   DropInserter.Drive.PLS.NotOperatorSide.HighLimit := 0.0;
   DropInserter.Drive.PLS.NotOperatorSide.Ok := FALSE;
   DropInserter.Drive.PLS.OnMould.LowLimit := 0.0;
   DropInserter.Drive.PLS.OnMould.HighLimit := 0.0;
   DropInserter.Drive.PLS.OnMould.Ok := FALSE;
   DropInserter.Drive.PLS.OffMould.LowLimit := 0.0;
   DropInserter.Drive.PLS.OffMould.HighLimit := 0.0;
   DropInserter.Drive.PLS.OffMould.Ok := FALSE;
   DropInserter.Drive.PLS.Pos0.LowLimit := 0.0;
   DropInserter.Drive.PLS.Pos0.HighLimit := 0.0;
   DropInserter.Drive.PLS.Pos0.Ok := FALSE;
   DropInserter.Drive.PLS.Pos1.LowLimit := 0.0;
   DropInserter.Drive.PLS.Pos1.HighLimit := 0.0;
   DropInserter.Drive.PLS.Pos1.Ok := FALSE;
   DropInserter.Drive.PLS.Pos2.LowLimit := 0.0;
   DropInserter.Drive.PLS.Pos2.HighLimit := 0.0;
   DropInserter.Drive.PLS.Pos2.Ok := FALSE;
   DropInserter.Drive.PLS.Pos3.LowLimit := 0.0;
   DropInserter.Drive.PLS.Pos3.HighLimit := 0.0;
   DropInserter.Drive.PLS.Pos3.Ok := FALSE;
   DropInserter.Drive.PLS.Pos4.LowLimit := 0.0;
   DropInserter.Drive.PLS.Pos4.HighLimit := 0.0;
   DropInserter.Drive.PLS.Pos4.Ok := FALSE;
   DropInserter.Drive.PLS.Pos5.LowLimit := 0.0;
   DropInserter.Drive.PLS.Pos5.HighLimit := 0.0;
   DropInserter.Drive.PLS.Pos5.Ok := FALSE;
   DropInserter.Drive.TON_EnableDrive.PT := T#500MS;
   DropInserter.Drive.TON_EnableDrive.IN := FALSE;
   DropInserter.Drive.TON_HwOvertravel_Dis.PT := T#0MS;
   DropInserter.Drive.TON_HwOvertravel_Dis.IN := FALSE;
   DropInserter.Drive.TON_HwOvertravel_En.PT := T#0MS;
   DropInserter.Drive.TON_HwOvertravel_En.IN := FALSE;
   DropInserter.Drive.TON_TimeoutMovement.PT := T#8S;
   DropInserter.Drive.TON_TimeoutMovement.IN := FALSE;
   DropInserter.TON_ResetMinLevel.PT := T#2S;
   DropInserter.TON_ResetMinLevel.IN := FALSE;
   DropInserter.RTO_Work.PT := T#1M;
   DropInserter.RTO_Work.IN := FALSE;
   DropInserter.TON_ScOK.PT := T#20S;
   DropInserter.TON_ScOK.IN := FALSE;
   DropInserter.TON_IncorrectPos.PT := T#2S;
   DropInserter.TON_IncorrectPos.IN := FALSE;
   DropInserter.TON_Sign_MinLevel.PT := T#1S;
   DropInserter.TON_Sign_MinLevel.IN := FALSE;
   DropInserter.TON_TimeoutWork.PT := T#20S;
   DropInserter.TON_TimeoutWork.IN := FALSE;
   DropInserter.TON_CloseCmd.PT := T#500MS;
   DropInserter.TON_CloseCmd.IN := FALSE;
   DropInserter.TON_MouldAbsence.PT := T#200MS;
   DropInserter.TON_MouldAbsence.IN := FALSE;
   PickInserter.ScOk := FALSE;
   PickInserter.CycleOn := FALSE;
   PickInserter.Work := FALSE;
   PickInserter.OkToStop := FALSE;
   PickInserter.AlmOk := TRUE;
   PickInserter.DrivesEnabled := FALSE;
   PickInserter.OutChainObstruction := FALSE;
   PickInserter.SingleCycle := FALSE;
   PickInserter.RepositioningReq := FALSE;
   PickInserter.Ons_TimeWork := FALSE;
   PickInserter.NumMinLevel := 0;
   PickInserter.Input.MouPreIns := FALSE;
   PickInserter.Input.EnaSel := FALSE;
   PickInserter.Input.MinLvl := FALSE;
   PickInserter.Input.HldCls := FALSE;
   PickInserter.Input.HldOpn := FALSE;
   PickInserter.Input.StrCls := FALSE;
   PickInserter.Input.StrOpn := FALSE;
   PickInserter.Output.EnaSelLgh := FALSE;
   PickInserter.Output.HldOpn := FALSE;
   PickInserter.Output.HldCls := FALSE;
   PickInserter.Output.StrOpn := FALSE;
   PickInserter.Output.StrCls := FALSE;
   PickInserter.Man.Ons_SingleCycle := FALSE;
   PickInserter.Man.CmdSupportOpen := FALSE;
   PickInserter.Man.CmdSupportClose := FALSE;
   PickInserter.Man.CmdStoreOpen := FALSE;
   PickInserter.Man.CmdStoreClose := FALSE;
   PickInserter.Man.CmdSingleCycle := FALSE;
   PickInserter.Man.EnaPbt := FALSE;
   PickInserter.Man.RstCmd := FALSE;
   PickInserter.Man.ScreenNumber := 302_080_301;
   PickInserter.Man.WithinScreenRange := 0;
   PickInserter."Step"._00_CycleActivated_DownCmd := FALSE;
   PickInserter."Step"._10_DownPos_OpenSupportCmd := FALSE;
   PickInserter."Step"._20_OpenSupportPos_CloseCmd := FALSE;
   PickInserter."Step"._30_ClosePos_CloseSupportCmd := FALSE;
   PickInserter."Step"._40_CloseSupportPos_UpCmd := FALSE;
   PickInserter."Step"._50_UpPos_OpenStoreCmd := FALSE;
   PickInserter."Step"._60_OpenStorePos_IntermediateCmd := FALSE;
   PickInserter."Step"._70_IntermediatePos_CloseStoreCmd := FALSE;
   PickInserter."Step"._80_CloseStorePos_CycleEnd := FALSE;
   PickInserter."Step".Ons_StrobeWorkDone := FALSE;
   PickInserter."Step".StrobeWorkDone := FALSE;
   PickInserter."Step".ScSeqOk := FALSE;
   PickInserter."Step".SeqActive := FALSE;
   PickInserter."Step".TON_WaitingHldOpn.PT := T#100MS;
   PickInserter."Step".TON_WaitingHldOpn.IN := FALSE;
   PickInserter."Step".TON_WaitingStrOpn.PT := T#100MS;
   PickInserter."Step".TON_WaitingStrOpn.IN := FALSE;
   PickInserter.Drive.AlmOk := FALSE;
   PickInserter.Drive.AlmEmerg := FALSE;
   PickInserter.Drive.AlmNode := FALSE;
   PickInserter.Drive.InitPosDrive := FALSE;
   PickInserter.Drive.InitPosDrivePLS := FALSE;
   PickInserter.Drive.GearingON := FALSE;
   PickInserter.Drive.CamHook := FALSE;
   PickInserter.Drive.CamStoppingPhase := FALSE;
   PickInserter.Drive.RepositioningRequest := FALSE;
   PickInserter.Drive.CamRequestResult := FALSE;
   PickInserter.Drive.CamRequestError := FALSE;
   PickInserter.Drive.CamRequestOk := FALSE;
   PickInserter.Drive.CalibDisAxisReq := FALSE;
   PickInserter.Drive.CalibReq := FALSE;
   PickInserter.Drive.CalibProcess := FALSE;
   PickInserter.Drive.HwOvertravelDisReq := FALSE;
   PickInserter.Drive.HwOvertravelEnReq := FALSE;
   PickInserter.Drive.AuxCamRequest := FALSE;
   PickInserter.Drive.TorquePeakEna := FALSE;
   PickInserter.Drive.Cmd_Repos := FALSE;
   PickInserter.Drive.Ons_CamRequest := FALSE;
   PickInserter.Drive.AuxCmdPosition := 0;
   PickInserter.Drive.Unwind := 0.0;
   PickInserter.Drive.MaxDev := 0.0;
   PickInserter.Drive.ReposSpeed := 100.0;
   PickInserter.Drive.CalcSlaveDifferenceABS := 0.0;
   PickInserter.Drive.CalcModPosition := 0.0;
   PickInserter.Drive.CalcSlaveDifference := 0.0;
   PickInserter.Drive.CalcMinDeltaPos := 0.0;
   PickInserter.Drive.CalcMaxDeltaPos := 0.0;
   PickInserter.Drive.CalcHalfPosUnwind := 0.0;
   PickInserter.Drive.Man.Cmd_PosJog := FALSE;
   PickInserter.Drive.Man.Cmd_NegJog := FALSE;
   PickInserter.Drive.Man.Cmd_Step := FALSE;
   PickInserter.Drive.Man.Cmd_Forward := FALSE;
   PickInserter.Drive.Man.Cmd_Backward := FALSE;
   PickInserter.Drive.Man.Cmd_Up := FALSE;
   PickInserter.Drive.Man.Cmd_Down := FALSE;
   PickInserter.Drive.Man.Cmd_Intermediate := FALSE;
   PickInserter.Drive.Man.Cmd_Open := FALSE;
   PickInserter.Drive.Man.Cmd_Close := FALSE;
   PickInserter.Drive.Man.Cmd_PreOpen := FALSE;
   PickInserter.Drive.Man.Cmd_Maintenance := FALSE;
   PickInserter.Drive.Man.Cmd_OperatorSide := FALSE;
   PickInserter.Drive.Man.Cmd_NotOperatorSide := FALSE;
   PickInserter.Drive.Man.Cmd_OnMould := FALSE;
   PickInserter.Drive.Man.Cmd_OffMould := FALSE;
   PickInserter.Drive.Man.Cmd_Pos0 := FALSE;
   PickInserter.Drive.Man.Cmd_Pos1 := FALSE;
   PickInserter.Drive.Man.Cmd_Pos2 := FALSE;
   PickInserter.Drive.Man.Cmd_Pos3 := FALSE;
   PickInserter.Drive.Man.Cmd_Pos4 := FALSE;
   PickInserter.Drive.Man.Cmd_Pos5 := FALSE;
   PickInserter.Drive.Man.Ons_Step := FALSE;
   PickInserter.Drive.Man.PhaseJogCmd := FALSE;
   PickInserter.Drive.Man.CmdStartStep := FALSE;
   PickInserter.Drive.Man.CmdEndStep := FALSE;
   PickInserter.Drive.Man.StepCond := FALSE;
   PickInserter.Drive.Man.TON_DelayHomeCmd.PT := T#3S;
   PickInserter.Drive.Man.TON_DelayHomeCmd.IN := FALSE;
   PickInserter.Drive.Auto.Cmd_Step := FALSE;
   PickInserter.Drive.Auto.Cmd_StartStep := FALSE;
   PickInserter.Drive.Auto.Cmd_EndStep := FALSE;
   PickInserter.Drive.Auto.Cmd_Forward := FALSE;
   PickInserter.Drive.Auto.Cmd_Backward := FALSE;
   PickInserter.Drive.Auto.Cmd_Up := FALSE;
   PickInserter.Drive.Auto.Cmd_Down := FALSE;
   PickInserter.Drive.Auto.Cmd_Intermediate := FALSE;
   PickInserter.Drive.Auto.Cmd_Open := FALSE;
   PickInserter.Drive.Auto.Cmd_Close := FALSE;
   PickInserter.Drive.Auto.Cmd_PreOpen := FALSE;
   PickInserter.Drive.Auto.Cmd_Maintenance := FALSE;
   PickInserter.Drive.Auto.Cmd_OperatorSide := FALSE;
   PickInserter.Drive.Auto.Cmd_NotOperatorSide := FALSE;
   PickInserter.Drive.Auto.Cmd_OnMould := FALSE;
   PickInserter.Drive.Auto.Cmd_OffMould := FALSE;
   PickInserter.Drive.Auto.Cmd_Pos0 := FALSE;
   PickInserter.Drive.Auto.Cmd_Pos1 := FALSE;
   PickInserter.Drive.Auto.Cmd_Pos2 := FALSE;
   PickInserter.Drive.Auto.Cmd_Pos3 := FALSE;
   PickInserter.Drive.Auto.Cmd_Pos4 := FALSE;
   PickInserter.Drive.Auto.Cmd_Pos5 := FALSE;
   PickInserter.Drive.Auto.Cmd_Gear := FALSE;
   PickInserter.Drive.ACT.CMD.Enable := FALSE;
   PickInserter.Drive.ACT.CMD.Pos_Mode := FALSE;
   PickInserter.Drive.ACT.CMD.MergeDisabled := FALSE;
   PickInserter.Drive.ACT.CMD.SCurve := FALSE;
   PickInserter.Drive.ACT.CMD.Cam_Mode := FALSE;
   PickInserter.Drive.ACT.CMD.Cam_Request := FALSE;
   PickInserter.Drive.ACT.CMD.Cam_PhaseStop := FALSE;
   PickInserter.Drive.ACT.CMD.Gear_Mode := FALSE;
   PickInserter.Drive.ACT.CMD.Repos_Req := FALSE;
   PickInserter.Drive.ACT.CMD.Jog_Pos := FALSE;
   PickInserter.Drive.ACT.CMD.Jog_Neg := FALSE;
   PickInserter.Drive.ACT.CMD.Stop := FALSE;
   PickInserter.Drive.ACT.CMD.Calibration_Req := FALSE;
   PickInserter.Drive.ACT.CMD.Reset := FALSE;
   PickInserter.Drive.ACT.CMD.RegInput1 := FALSE;
   PickInserter.Drive.ACT.CMD.Brake_Release := FALSE;
   PickInserter.Drive.ACT.CMD.HwPosOvertravel_Dis := FALSE;
   PickInserter.Drive.ACT.CMD.HwNegOvertravel_Dis := FALSE;
   PickInserter.Drive.ACT.CMD.HwOvertravel_MSG_En := FALSE;
   PickInserter.Drive.ACT.CMD.OneShootMove := FALSE;
   PickInserter.Drive.ACT.CMD.Move_Type := 0;
   PickInserter.Drive.ACT.CMD.Target_Pos := 0.0;
   PickInserter.Drive.ACT.CMD.Speed := 0.0;
   PickInserter.Drive.ACT.CMD.Acceleration := 0.0;
   PickInserter.Drive.ACT.CMD.Deceleration := 0.0;
   PickInserter.Drive.ACT.CMD.Torque_Limit := 0.0;
   PickInserter.Drive.ACT.CMD.Gear_Ratio := 0.0;
   PickInserter.Drive.ACT.CMD.Mccp_Length := 0;
   PickInserter.Drive.ACT.CMD.Mccp_StartSlope := 0.0;
   PickInserter.Drive.ACT.CMD.Mccp_EndSlope := 0.0;
   PickInserter.Drive.ACT.CMD.Mapc_Direction := 0;
   PickInserter.Drive.ACT.CMD.Mapc_SlaveScaling := 0.0;
   PickInserter.Drive.ACT.CMD.Mapc_MasterScaling := 0.0;
   PickInserter.Drive.ACT.CMD.Mapc_MasterLockPosition := 0.0;
   PickInserter.Drive.ACT.CMD.Mapc_CamLockPosition := 0.0;
   PickInserter.Drive.ACT.CMD.Cam[0..39].leadingValueStart := 0.0;
   PickInserter.Drive.ACT.CMD.Cam[0..39].leadingValueEnd := 0.0;
   PickInserter.Drive.ACT.CMD.Cam[0..39].followingValueStart := 0.0;
   PickInserter.Drive.ACT.CMD.Cam[0..39].followingValueEnd := 0.0;
   PickInserter.Drive.ACT.CMD.Cam[0..39].geoVeloStart := 0.0;
   PickInserter.Drive.ACT.CMD.Cam[0..39].geoVeloEnd := 0.0;
   PickInserter.Drive.ACT.CMD.Cam[0..39].geoAccelStart := 0.0;
   PickInserter.Drive.ACT.CMD.Cam[0..39].geoAccelEnd := 0.0;
   PickInserter.Drive.ACT.CMD.Cam[0..39].geoJerkStart := 0.0;
   PickInserter.Drive.ACT.CMD.Cam[0..39].geoJerkEnd := 0.0;
   PickInserter.Drive.ACT.CMD.Cam[0..39].inflectionPointParameter := 0.5;
   PickInserter.Drive.ACT.CMD.Cam[0..39].modVeloTrapezoidParameter := 1.0;
   PickInserter.Drive.ACT.CMD.Cam[0..39].modSineMaxAccelCaStar := 0.0;
   PickInserter.Drive.ACT.CMD.Cam[0..39].camProfileType := 0;
   PickInserter.Drive.ACT.FBK.Ready := FALSE;
   PickInserter.Drive.ACT.FBK.Calibrated := FALSE;
   PickInserter.Drive.ACT.FBK.Fault := FALSE;
   PickInserter.Drive.ACT.FBK.ModuleConnFault := FALSE;
   PickInserter.Drive.ACT.FBK.In_Position := FALSE;
   PickInserter.Drive.ACT.FBK.Standstill := FALSE;
   PickInserter.Drive.ACT.FBK.Enabled := FALSE;
   PickInserter.Drive.ACT.FBK.BusReadyStatus := FALSE;
   PickInserter.Drive.ACT.FBK.BrakeReleased := FALSE;
   PickInserter.Drive.ACT.FBK.HwPosOvertravelDisabled := FALSE;
   PickInserter.Drive.ACT.FBK.HwNegOvertravelDisabled := FALSE;
   PickInserter.Drive.ACT.FBK.SafeOffStatus := FALSE;
   PickInserter.Drive.ACT.FBK.MaxTorqueLimit := FALSE;
   PickInserter.Drive.ACT.FBK.PosMerge_IP := FALSE;
   PickInserter.Drive.ACT.FBK.PosMerge_PC := FALSE;
   PickInserter.Drive.ACT.FBK.Gearing_IP := FALSE;
   PickInserter.Drive.ACT.FBK.Position := 0.0;
   PickInserter.Drive.ACT.FBK.Speed := 0.0;
   PickInserter.Drive.ACT.FBK.Torque := 0.0;
   PickInserter.Drive.ACT.FBK.RegInput1Pos := 0.0;
   PickInserter.Drive.ACT.FBK.SeqCamErrorCode := 0;
   PickInserter.Drive.ACT.FBK.SeqCamTargetPosMAM := 0.0;
   PickInserter.Drive.ACT.FBK.SeqCamStatus.EndSequence := FALSE;
   PickInserter.Drive.ACT.FBK.SeqCamStatus.EndSuccess := FALSE;
   PickInserter.Drive.ACT.FBK.SeqCamStatus.EndError := FALSE;
   PickInserter.Drive.ACT.FBK.SeqCamStatus.CamHook := FALSE;
   PickInserter.Drive.ACT.FBK.SeqCamStatus.BothMapc_IP := FALSE;
   PickInserter.Drive.ACT.FBK.SeqCamStatus.SlaveFwd := FALSE;
   PickInserter.Drive.ACT.FBK.SeqCamStatus.SlaveBwd := FALSE;
   PickInserter.Drive.ACT.FBK.SeqCamStatus.SlaveUnwind := FALSE;
   PickInserter.Drive.ACT.FBK.SeqCamStatus.WaitValidByOpe := FALSE;
   PickInserter.Drive.ACT.FBK.SeqCamStatus.MapcA_IP := FALSE;
   PickInserter.Drive.ACT.FBK.SeqCamStatus.MapcB_IP := FALSE;
   PickInserter.Drive.ACT.FBK.SeqCamStatus.MapcC_IP := FALSE;
   PickInserter.Drive.ACT.FBK.SeqCamStatus.CamOnce_PC := FALSE;
   PickInserter.Drive.ACT.FBK.SeqCamStatus.MaxDevError := FALSE;
   PickInserter.Drive.ACT.FBK.SeqCamStatus.PositionCamLockStatus := FALSE;
   PickInserter.Drive.ACT.FBK.SeqCamStatus.WaitRestart := FALSE;
   PickInserter.Drive.ACT.FBK.SeqCamStatus.Bit17 := FALSE;
   PickInserter.Drive.ACT.FBK.SeqCamStatus.Bit18 := FALSE;
   PickInserter.Drive.ACT.FBK.SeqCamStatus.Bit19 := FALSE;
   PickInserter.Drive.ACT.FBK.SeqCamStatus.Bit20 := FALSE;
   PickInserter.Drive.ACT.FBK.SeqCamStatus.Bit21 := FALSE;
   PickInserter.Drive.ACT.FBK.SeqCamStatus.Bit22 := FALSE;
   PickInserter.Drive.ACT.FBK.SeqCamStatus.Bit23 := FALSE;
   PickInserter.Drive.ACT.FBK.SeqCamStatus.Bit24 := FALSE;
   PickInserter.Drive.ACT.FBK.SeqCamStatus.Bit25 := FALSE;
   PickInserter.Drive.ACT.FBK.SeqCamStatus.Bit26 := FALSE;
   PickInserter.Drive.ACT.FBK.SeqCamStatus.Bit27 := FALSE;
   PickInserter.Drive.ACT.FBK.SeqCamStatus.Bit28 := FALSE;
   PickInserter.Drive.ACT.FBK.SeqCamStatus.Bit29 := FALSE;
   PickInserter.Drive.ACT.FBK.SeqCamStatus.Bit30 := FALSE;
   PickInserter.Drive.ACT.FBK.SeqCamStatus.Bit31 := FALSE;
   PickInserter.Drive.ACT.FBK.SeqCamStatus.Bit32 := FALSE;
   PickInserter.Drive.PLS.FinePosOk.LowLimit := 0.0;
   PickInserter.Drive.PLS.FinePosOk.HighLimit := 0.0;
   PickInserter.Drive.PLS.FinePosOk.Ok := FALSE;
   PickInserter.Drive.PLS.KeepPosOk.LowLimit := 0.0;
   PickInserter.Drive.PLS.KeepPosOk.HighLimit := 0.0;
   PickInserter.Drive.PLS.KeepPosOk.Ok := FALSE;
   PickInserter.Drive.PLS.Up.LowLimit := 0.0;
   PickInserter.Drive.PLS.Up.HighLimit := 0.0;
   PickInserter.Drive.PLS.Up.Ok := FALSE;
   PickInserter.Drive.PLS.Intermediate.LowLimit := 0.0;
   PickInserter.Drive.PLS.Intermediate.HighLimit := 0.0;
   PickInserter.Drive.PLS.Intermediate.Ok := FALSE;
   PickInserter.Drive.PLS.Down.LowLimit := 0.0;
   PickInserter.Drive.PLS.Down.HighLimit := 0.0;
   PickInserter.Drive.PLS.Down.Ok := FALSE;
   PickInserter.Drive.PLS.Forward.LowLimit := 0.0;
   PickInserter.Drive.PLS.Forward.HighLimit := 0.0;
   PickInserter.Drive.PLS.Forward.Ok := FALSE;
   PickInserter.Drive.PLS.Backward.LowLimit := 0.0;
   PickInserter.Drive.PLS.Backward.HighLimit := 0.0;
   PickInserter.Drive.PLS.Backward.Ok := FALSE;
   PickInserter.Drive.PLS.Open.LowLimit := 0.0;
   PickInserter.Drive.PLS.Open.HighLimit := 0.0;
   PickInserter.Drive.PLS.Open.Ok := FALSE;
   PickInserter.Drive.PLS.Close.LowLimit := 0.0;
   PickInserter.Drive.PLS.Close.HighLimit := 0.0;
   PickInserter.Drive.PLS.Close.Ok := FALSE;
   PickInserter.Drive.PLS.PreOpen.LowLimit := 0.0;
   PickInserter.Drive.PLS.PreOpen.HighLimit := 0.0;
   PickInserter.Drive.PLS.PreOpen.Ok := FALSE;
   PickInserter.Drive.PLS.Maintenance.LowLimit := 0.0;
   PickInserter.Drive.PLS.Maintenance.HighLimit := 0.0;
   PickInserter.Drive.PLS.Maintenance.Ok := FALSE;
   PickInserter.Drive.PLS.OperatorSide.LowLimit := 0.0;
   PickInserter.Drive.PLS.OperatorSide.HighLimit := 0.0;
   PickInserter.Drive.PLS.OperatorSide.Ok := FALSE;
   PickInserter.Drive.PLS.NotOperatorSide.LowLimit := 0.0;
   PickInserter.Drive.PLS.NotOperatorSide.HighLimit := 0.0;
   PickInserter.Drive.PLS.NotOperatorSide.Ok := FALSE;
   PickInserter.Drive.PLS.OnMould.LowLimit := 0.0;
   PickInserter.Drive.PLS.OnMould.HighLimit := 0.0;
   PickInserter.Drive.PLS.OnMould.Ok := FALSE;
   PickInserter.Drive.PLS.OffMould.LowLimit := 0.0;
   PickInserter.Drive.PLS.OffMould.HighLimit := 0.0;
   PickInserter.Drive.PLS.OffMould.Ok := FALSE;
   PickInserter.Drive.PLS.Pos0.LowLimit := 0.0;
   PickInserter.Drive.PLS.Pos0.HighLimit := 0.0;
   PickInserter.Drive.PLS.Pos0.Ok := FALSE;
   PickInserter.Drive.PLS.Pos1.LowLimit := 0.0;
   PickInserter.Drive.PLS.Pos1.HighLimit := 0.0;
   PickInserter.Drive.PLS.Pos1.Ok := FALSE;
   PickInserter.Drive.PLS.Pos2.LowLimit := 0.0;
   PickInserter.Drive.PLS.Pos2.HighLimit := 0.0;
   PickInserter.Drive.PLS.Pos2.Ok := FALSE;
   PickInserter.Drive.PLS.Pos3.LowLimit := 0.0;
   PickInserter.Drive.PLS.Pos3.HighLimit := 0.0;
   PickInserter.Drive.PLS.Pos3.Ok := FALSE;
   PickInserter.Drive.PLS.Pos4.LowLimit := 0.0;
   PickInserter.Drive.PLS.Pos4.HighLimit := 0.0;
   PickInserter.Drive.PLS.Pos4.Ok := FALSE;
   PickInserter.Drive.PLS.Pos5.LowLimit := 0.0;
   PickInserter.Drive.PLS.Pos5.HighLimit := 0.0;
   PickInserter.Drive.PLS.Pos5.Ok := FALSE;
   PickInserter.Drive.TON_EnableDrive.PT := T#500MS;
   PickInserter.Drive.TON_EnableDrive.IN := FALSE;
   PickInserter.Drive.TON_HwOvertravel_Dis.PT := T#0MS;
   PickInserter.Drive.TON_HwOvertravel_Dis.IN := FALSE;
   PickInserter.Drive.TON_HwOvertravel_En.PT := T#0MS;
   PickInserter.Drive.TON_HwOvertravel_En.IN := FALSE;
   PickInserter.Drive.TON_TimeoutMovement.PT := T#8S;
   PickInserter.Drive.TON_TimeoutMovement.IN := FALSE;
   PickInserter.TON_ResetMinLevel.PT := T#2S;
   PickInserter.TON_ResetMinLevel.IN := FALSE;
   PickInserter.RTO_Work.PT := T#1M;
   PickInserter.RTO_Work.IN := FALSE;
   PickInserter.TON_ScOK.PT := T#20S;
   PickInserter.TON_ScOK.IN := FALSE;
   PickInserter.TON_SupportIncorrectPos.PT := T#2S;
   PickInserter.TON_SupportIncorrectPos.IN := FALSE;
   PickInserter.TON_StoreIncorrectPos.PT := T#2S;
   PickInserter.TON_StoreIncorrectPos.IN := FALSE;
   PickInserter.TON_Sign_MinLevel.PT := T#1S;
   PickInserter.TON_Sign_MinLevel.IN := FALSE;
   PickInserter.TON_TimeoutWork.PT := T#20S;
   PickInserter.TON_TimeoutWork.IN := FALSE;
   PickInserter.TON_MouldAbsence.PT := T#200MS;
   PickInserter.TON_MouldAbsence.IN := FALSE;
   RotaryInserter.ScOk := FALSE;
   RotaryInserter.CycleOn := FALSE;
   RotaryInserter.Work := FALSE;
   RotaryInserter.OkToStop := TRUE;
   RotaryInserter.AlmOk := TRUE;
   RotaryInserter.DrivesEnabled := FALSE;
   RotaryInserter.OutChainObstruction := TRUE;
   RotaryInserter.RepositioningReq := FALSE;
   RotaryInserter.Ons_TimeWork := TRUE;
   RotaryInserter.NumMinLevel := 0;
   RotaryInserter.Input.MouPreIns := TRUE;
   RotaryInserter.Input.EnaSel := FALSE;
   RotaryInserter.Input.MinLvl := TRUE;
   RotaryInserter.Output.EnaSelLgh := FALSE;
   RotaryInserter.Man.EnaPbt := FALSE;
   RotaryInserter.Man.RstCmd := TRUE;
   RotaryInserter.Man.ScreenNumber := 302_090_301;
   RotaryInserter.Man.WithinScreenRange := 0;
   RotaryInserter."Step"._00_CycleActived_StartRotationCmd := FALSE;
   RotaryInserter."Step"._10_RotationOutPos_StopRotationCmd := FALSE;
   RotaryInserter."Step"._20_FinePos_IncreaseMinLevMouCmd := FALSE;
   RotaryInserter."Step"._30_MinLevInc_CycleEnd := FALSE;
   RotaryInserter."Step".Ons_StrobeWorkDone := FALSE;
   RotaryInserter."Step".StrobeWorkDone := FALSE;
   RotaryInserter."Step".ScSeqOk := FALSE;
   RotaryInserter."Step".SeqActive := FALSE;
   RotaryInserter.Drive.AlmOk := FALSE;
   RotaryInserter.Drive.AlmEmerg := FALSE;
   RotaryInserter.Drive.AlmNode := FALSE;
   RotaryInserter.Drive.InitPosDrive := FALSE;
   RotaryInserter.Drive.InitPosDrivePLS := FALSE;
   RotaryInserter.Drive.GearingON := FALSE;
   RotaryInserter.Drive.CamHook := FALSE;
   RotaryInserter.Drive.CamStoppingPhase := FALSE;
   RotaryInserter.Drive.RepositioningRequest := FALSE;
   RotaryInserter.Drive.CamRequestResult := FALSE;
   RotaryInserter.Drive.CamRequestError := FALSE;
   RotaryInserter.Drive.CamRequestOk := FALSE;
   RotaryInserter.Drive.CalibDisAxisReq := FALSE;
   RotaryInserter.Drive.CalibReq := FALSE;
   RotaryInserter.Drive.CalibProcess := FALSE;
   RotaryInserter.Drive.HwOvertravelDisReq := FALSE;
   RotaryInserter.Drive.HwOvertravelEnReq := FALSE;
   RotaryInserter.Drive.AuxCamRequest := FALSE;
   RotaryInserter.Drive.TorquePeakEna := TRUE;
   RotaryInserter.Drive.Cmd_Repos := FALSE;
   RotaryInserter.Drive.Ons_CamRequest := FALSE;
   RotaryInserter.Drive.AuxCmdPosition := 0;
   RotaryInserter.Drive.Unwind := 360.0;
   RotaryInserter.Drive.MaxDev := 0.0;
   RotaryInserter.Drive.ReposSpeed := 100.0;
   RotaryInserter.Drive.CalcSlaveDifferenceABS := 0.0;
   RotaryInserter.Drive.CalcModPosition := 0.0;
   RotaryInserter.Drive.CalcSlaveDifference := 0.0;
   RotaryInserter.Drive.CalcMinDeltaPos := 0.0;
   RotaryInserter.Drive.CalcMaxDeltaPos := 0.0;
   RotaryInserter.Drive.CalcHalfPosUnwind := 0.0;
   RotaryInserter.Drive.Man.Cmd_PosJog := FALSE;
   RotaryInserter.Drive.Man.Cmd_NegJog := FALSE;
   RotaryInserter.Drive.Man.Cmd_Step := FALSE;
   RotaryInserter.Drive.Man.Cmd_Forward := FALSE;
   RotaryInserter.Drive.Man.Cmd_Backward := FALSE;
   RotaryInserter.Drive.Man.Cmd_Up := FALSE;
   RotaryInserter.Drive.Man.Cmd_Down := FALSE;
   RotaryInserter.Drive.Man.Cmd_Intermediate := FALSE;
   RotaryInserter.Drive.Man.Cmd_Open := FALSE;
   RotaryInserter.Drive.Man.Cmd_Close := FALSE;
   RotaryInserter.Drive.Man.Cmd_PreOpen := FALSE;
   RotaryInserter.Drive.Man.Cmd_Maintenance := FALSE;
   RotaryInserter.Drive.Man.Cmd_OperatorSide := FALSE;
   RotaryInserter.Drive.Man.Cmd_NotOperatorSide := FALSE;
   RotaryInserter.Drive.Man.Cmd_OnMould := FALSE;
   RotaryInserter.Drive.Man.Cmd_OffMould := FALSE;
   RotaryInserter.Drive.Man.Cmd_Pos0 := FALSE;
   RotaryInserter.Drive.Man.Cmd_Pos1 := FALSE;
   RotaryInserter.Drive.Man.Cmd_Pos2 := FALSE;
   RotaryInserter.Drive.Man.Cmd_Pos3 := FALSE;
   RotaryInserter.Drive.Man.Cmd_Pos4 := FALSE;
   RotaryInserter.Drive.Man.Cmd_Pos5 := FALSE;
   RotaryInserter.Drive.Man.Ons_Step := FALSE;
   RotaryInserter.Drive.Man.PhaseJogCmd := FALSE;
   RotaryInserter.Drive.Man.CmdStartStep := FALSE;
   RotaryInserter.Drive.Man.CmdEndStep := FALSE;
   RotaryInserter.Drive.Man.StepCond := FALSE;
   RotaryInserter.Drive.Man.TON_DelayHomeCmd.PT := T#3S;
   RotaryInserter.Drive.Man.TON_DelayHomeCmd.IN := FALSE;
   RotaryInserter.Drive.Auto.Cmd_Step := FALSE;
   RotaryInserter.Drive.Auto.Cmd_StartStep := FALSE;
   RotaryInserter.Drive.Auto.Cmd_EndStep := FALSE;
   RotaryInserter.Drive.Auto.Cmd_Forward := FALSE;
   RotaryInserter.Drive.Auto.Cmd_Backward := FALSE;
   RotaryInserter.Drive.Auto.Cmd_Up := FALSE;
   RotaryInserter.Drive.Auto.Cmd_Down := FALSE;
   RotaryInserter.Drive.Auto.Cmd_Intermediate := FALSE;
   RotaryInserter.Drive.Auto.Cmd_Open := FALSE;
   RotaryInserter.Drive.Auto.Cmd_Close := FALSE;
   RotaryInserter.Drive.Auto.Cmd_PreOpen := FALSE;
   RotaryInserter.Drive.Auto.Cmd_Maintenance := FALSE;
   RotaryInserter.Drive.Auto.Cmd_OperatorSide := FALSE;
   RotaryInserter.Drive.Auto.Cmd_NotOperatorSide := FALSE;
   RotaryInserter.Drive.Auto.Cmd_OnMould := FALSE;
   RotaryInserter.Drive.Auto.Cmd_OffMould := FALSE;
   RotaryInserter.Drive.Auto.Cmd_Pos0 := FALSE;
   RotaryInserter.Drive.Auto.Cmd_Pos1 := FALSE;
   RotaryInserter.Drive.Auto.Cmd_Pos2 := FALSE;
   RotaryInserter.Drive.Auto.Cmd_Pos3 := FALSE;
   RotaryInserter.Drive.Auto.Cmd_Pos4 := FALSE;
   RotaryInserter.Drive.Auto.Cmd_Pos5 := FALSE;
   RotaryInserter.Drive.Auto.Cmd_Gear := FALSE;
   RotaryInserter.Drive.ACT.CMD.Enable := FALSE;
   RotaryInserter.Drive.ACT.CMD.Pos_Mode := FALSE;
   RotaryInserter.Drive.ACT.CMD.MergeDisabled := FALSE;
   RotaryInserter.Drive.ACT.CMD.SCurve := FALSE;
   RotaryInserter.Drive.ACT.CMD.Cam_Mode := FALSE;
   RotaryInserter.Drive.ACT.CMD.Cam_Request := FALSE;
   RotaryInserter.Drive.ACT.CMD.Cam_PhaseStop := FALSE;
   RotaryInserter.Drive.ACT.CMD.Gear_Mode := FALSE;
   RotaryInserter.Drive.ACT.CMD.Repos_Req := FALSE;
   RotaryInserter.Drive.ACT.CMD.Jog_Pos := FALSE;
   RotaryInserter.Drive.ACT.CMD.Jog_Neg := FALSE;
   RotaryInserter.Drive.ACT.CMD.Stop := TRUE;
   RotaryInserter.Drive.ACT.CMD.Calibration_Req := FALSE;
   RotaryInserter.Drive.ACT.CMD.Reset := FALSE;
   RotaryInserter.Drive.ACT.CMD.RegInput1 := FALSE;
   RotaryInserter.Drive.ACT.CMD.Brake_Release := FALSE;
   RotaryInserter.Drive.ACT.CMD.HwPosOvertravel_Dis := FALSE;
   RotaryInserter.Drive.ACT.CMD.HwNegOvertravel_Dis := FALSE;
   RotaryInserter.Drive.ACT.CMD.HwOvertravel_MSG_En := FALSE;
   RotaryInserter.Drive.ACT.CMD.OneShootMove := FALSE;
   RotaryInserter.Drive.ACT.CMD.Move_Type := 3;
   RotaryInserter.Drive.ACT.CMD.Target_Pos := 0.0;
   RotaryInserter.Drive.ACT.CMD.Speed := 250.0;
   RotaryInserter.Drive.ACT.CMD.Acceleration := 4000.0;
   RotaryInserter.Drive.ACT.CMD.Deceleration := 4500.0;
   RotaryInserter.Drive.ACT.CMD.Torque_Limit := 50.0;
   RotaryInserter.Drive.ACT.CMD.Gear_Ratio := 0.0;
   RotaryInserter.Drive.ACT.CMD.Mccp_Length := 0;
   RotaryInserter.Drive.ACT.CMD.Mccp_StartSlope := 0.0;
   RotaryInserter.Drive.ACT.CMD.Mccp_EndSlope := 0.0;
   RotaryInserter.Drive.ACT.CMD.Mapc_Direction := 0;
   RotaryInserter.Drive.ACT.CMD.Mapc_SlaveScaling := 0.0;
   RotaryInserter.Drive.ACT.CMD.Mapc_MasterScaling := 0.0;
   RotaryInserter.Drive.ACT.CMD.Mapc_MasterLockPosition := 0.0;
   RotaryInserter.Drive.ACT.CMD.Mapc_CamLockPosition := 0.0;
   RotaryInserter.Drive.ACT.CMD.Cam[0..39].leadingValueStart := 0.0;
   RotaryInserter.Drive.ACT.CMD.Cam[0..39].leadingValueEnd := 0.0;
   RotaryInserter.Drive.ACT.CMD.Cam[0..39].followingValueStart := 0.0;
   RotaryInserter.Drive.ACT.CMD.Cam[0..39].followingValueEnd := 0.0;
   RotaryInserter.Drive.ACT.CMD.Cam[0..39].geoVeloStart := 0.0;
   RotaryInserter.Drive.ACT.CMD.Cam[0..39].geoVeloEnd := 0.0;
   RotaryInserter.Drive.ACT.CMD.Cam[0..39].geoAccelStart := 0.0;
   RotaryInserter.Drive.ACT.CMD.Cam[0..39].geoAccelEnd := 0.0;
   RotaryInserter.Drive.ACT.CMD.Cam[0..39].geoJerkStart := 0.0;
   RotaryInserter.Drive.ACT.CMD.Cam[0..39].geoJerkEnd := 0.0;
   RotaryInserter.Drive.ACT.CMD.Cam[0..39].inflectionPointParameter := 0.5;
   RotaryInserter.Drive.ACT.CMD.Cam[0..39].modVeloTrapezoidParameter := 1.0;
   RotaryInserter.Drive.ACT.CMD.Cam[0..39].modSineMaxAccelCaStar := 0.0;
   RotaryInserter.Drive.ACT.CMD.Cam[0..39].camProfileType := 0;
   RotaryInserter.Drive.ACT.FBK.Ready := TRUE;
   RotaryInserter.Drive.ACT.FBK.Calibrated := TRUE;
   RotaryInserter.Drive.ACT.FBK.Fault := FALSE;
   RotaryInserter.Drive.ACT.FBK.ModuleConnFault := FALSE;
   RotaryInserter.Drive.ACT.FBK.In_Position := FALSE;
   RotaryInserter.Drive.ACT.FBK.Standstill := TRUE;
   RotaryInserter.Drive.ACT.FBK.Enabled := FALSE;
   RotaryInserter.Drive.ACT.FBK.BusReadyStatus := FALSE;
   RotaryInserter.Drive.ACT.FBK.BrakeReleased := FALSE;
   RotaryInserter.Drive.ACT.FBK.HwPosOvertravelDisabled := FALSE;
   RotaryInserter.Drive.ACT.FBK.HwNegOvertravelDisabled := FALSE;
   RotaryInserter.Drive.ACT.FBK.SafeOffStatus := FALSE;
   RotaryInserter.Drive.ACT.FBK.MaxTorqueLimit := FALSE;
   RotaryInserter.Drive.ACT.FBK.PosMerge_IP := FALSE;
   RotaryInserter.Drive.ACT.FBK.PosMerge_PC := FALSE;
   RotaryInserter.Drive.ACT.FBK.Gearing_IP := FALSE;
   RotaryInserter.Drive.ACT.FBK.Position := 0.81;
   RotaryInserter.Drive.ACT.FBK.Speed := -0.02503395;
   RotaryInserter.Drive.ACT.FBK.Torque := 0.0;
   RotaryInserter.Drive.ACT.FBK.RegInput1Pos := 0.0;
   RotaryInserter.Drive.ACT.FBK.SeqCamErrorCode := 0;
   RotaryInserter.Drive.ACT.FBK.SeqCamTargetPosMAM := 0.0;
   RotaryInserter.Drive.ACT.FBK.SeqCamStatus.EndSequence := FALSE;
   RotaryInserter.Drive.ACT.FBK.SeqCamStatus.EndSuccess := FALSE;
   RotaryInserter.Drive.ACT.FBK.SeqCamStatus.EndError := FALSE;
   RotaryInserter.Drive.ACT.FBK.SeqCamStatus.CamHook := FALSE;
   RotaryInserter.Drive.ACT.FBK.SeqCamStatus.BothMapc_IP := FALSE;
   RotaryInserter.Drive.ACT.FBK.SeqCamStatus.SlaveFwd := FALSE;
   RotaryInserter.Drive.ACT.FBK.SeqCamStatus.SlaveBwd := FALSE;
   RotaryInserter.Drive.ACT.FBK.SeqCamStatus.SlaveUnwind := FALSE;
   RotaryInserter.Drive.ACT.FBK.SeqCamStatus.WaitValidByOpe := FALSE;
   RotaryInserter.Drive.ACT.FBK.SeqCamStatus.MapcA_IP := FALSE;
   RotaryInserter.Drive.ACT.FBK.SeqCamStatus.MapcB_IP := FALSE;
   RotaryInserter.Drive.ACT.FBK.SeqCamStatus.MapcC_IP := FALSE;
   RotaryInserter.Drive.ACT.FBK.SeqCamStatus.CamOnce_PC := FALSE;
   RotaryInserter.Drive.ACT.FBK.SeqCamStatus.MaxDevError := FALSE;
   RotaryInserter.Drive.ACT.FBK.SeqCamStatus.PositionCamLockStatus := FALSE;
   RotaryInserter.Drive.ACT.FBK.SeqCamStatus.WaitRestart := FALSE;
   RotaryInserter.Drive.ACT.FBK.SeqCamStatus.Bit17 := FALSE;
   RotaryInserter.Drive.ACT.FBK.SeqCamStatus.Bit18 := FALSE;
   RotaryInserter.Drive.ACT.FBK.SeqCamStatus.Bit19 := FALSE;
   RotaryInserter.Drive.ACT.FBK.SeqCamStatus.Bit20 := FALSE;
   RotaryInserter.Drive.ACT.FBK.SeqCamStatus.Bit21 := FALSE;
   RotaryInserter.Drive.ACT.FBK.SeqCamStatus.Bit22 := FALSE;
   RotaryInserter.Drive.ACT.FBK.SeqCamStatus.Bit23 := FALSE;
   RotaryInserter.Drive.ACT.FBK.SeqCamStatus.Bit24 := FALSE;
   RotaryInserter.Drive.ACT.FBK.SeqCamStatus.Bit25 := FALSE;
   RotaryInserter.Drive.ACT.FBK.SeqCamStatus.Bit26 := FALSE;
   RotaryInserter.Drive.ACT.FBK.SeqCamStatus.Bit27 := FALSE;
   RotaryInserter.Drive.ACT.FBK.SeqCamStatus.Bit28 := FALSE;
   RotaryInserter.Drive.ACT.FBK.SeqCamStatus.Bit29 := FALSE;
   RotaryInserter.Drive.ACT.FBK.SeqCamStatus.Bit30 := FALSE;
   RotaryInserter.Drive.ACT.FBK.SeqCamStatus.Bit31 := FALSE;
   RotaryInserter.Drive.ACT.FBK.SeqCamStatus.Bit32 := FALSE;
   RotaryInserter.Drive.PLS.FinePosOk.LowLimit := 357.0;
   RotaryInserter.Drive.PLS.FinePosOk.HighLimit := 3.0;
   RotaryInserter.Drive.PLS.FinePosOk.Ok := TRUE;
   RotaryInserter.Drive.PLS.KeepPosOk.LowLimit := 0.0;
   RotaryInserter.Drive.PLS.KeepPosOk.HighLimit := 0.0;
   RotaryInserter.Drive.PLS.KeepPosOk.Ok := FALSE;
   RotaryInserter.Drive.PLS.Up.LowLimit := 0.0;
   RotaryInserter.Drive.PLS.Up.HighLimit := 0.0;
   RotaryInserter.Drive.PLS.Up.Ok := FALSE;
   RotaryInserter.Drive.PLS.Intermediate.LowLimit := 0.0;
   RotaryInserter.Drive.PLS.Intermediate.HighLimit := 0.0;
   RotaryInserter.Drive.PLS.Intermediate.Ok := FALSE;
   RotaryInserter.Drive.PLS.Down.LowLimit := 0.0;
   RotaryInserter.Drive.PLS.Down.HighLimit := 0.0;
   RotaryInserter.Drive.PLS.Down.Ok := FALSE;
   RotaryInserter.Drive.PLS.Forward.LowLimit := 0.0;
   RotaryInserter.Drive.PLS.Forward.HighLimit := 0.0;
   RotaryInserter.Drive.PLS.Forward.Ok := FALSE;
   RotaryInserter.Drive.PLS.Backward.LowLimit := 0.0;
   RotaryInserter.Drive.PLS.Backward.HighLimit := 0.0;
   RotaryInserter.Drive.PLS.Backward.Ok := FALSE;
   RotaryInserter.Drive.PLS.Open.LowLimit := 0.0;
   RotaryInserter.Drive.PLS.Open.HighLimit := 0.0;
   RotaryInserter.Drive.PLS.Open.Ok := FALSE;
   RotaryInserter.Drive.PLS.Close.LowLimit := 0.0;
   RotaryInserter.Drive.PLS.Close.HighLimit := 0.0;
   RotaryInserter.Drive.PLS.Close.Ok := FALSE;
   RotaryInserter.Drive.PLS.PreOpen.LowLimit := 0.0;
   RotaryInserter.Drive.PLS.PreOpen.HighLimit := 0.0;
   RotaryInserter.Drive.PLS.PreOpen.Ok := FALSE;
   RotaryInserter.Drive.PLS.Maintenance.LowLimit := 0.0;
   RotaryInserter.Drive.PLS.Maintenance.HighLimit := 0.0;
   RotaryInserter.Drive.PLS.Maintenance.Ok := FALSE;
   RotaryInserter.Drive.PLS.OperatorSide.LowLimit := 0.0;
   RotaryInserter.Drive.PLS.OperatorSide.HighLimit := 0.0;
   RotaryInserter.Drive.PLS.OperatorSide.Ok := FALSE;
   RotaryInserter.Drive.PLS.NotOperatorSide.LowLimit := 0.0;
   RotaryInserter.Drive.PLS.NotOperatorSide.HighLimit := 0.0;
   RotaryInserter.Drive.PLS.NotOperatorSide.Ok := FALSE;
   RotaryInserter.Drive.PLS.OnMould.LowLimit := 0.0;
   RotaryInserter.Drive.PLS.OnMould.HighLimit := 0.0;
   RotaryInserter.Drive.PLS.OnMould.Ok := FALSE;
   RotaryInserter.Drive.PLS.OffMould.LowLimit := 0.0;
   RotaryInserter.Drive.PLS.OffMould.HighLimit := 0.0;
   RotaryInserter.Drive.PLS.OffMould.Ok := FALSE;
   RotaryInserter.Drive.PLS.Pos0.LowLimit := 0.0;
   RotaryInserter.Drive.PLS.Pos0.HighLimit := 0.0;
   RotaryInserter.Drive.PLS.Pos0.Ok := FALSE;
   RotaryInserter.Drive.PLS.Pos1.LowLimit := 0.0;
   RotaryInserter.Drive.PLS.Pos1.HighLimit := 0.0;
   RotaryInserter.Drive.PLS.Pos1.Ok := FALSE;
   RotaryInserter.Drive.PLS.Pos2.LowLimit := 0.0;
   RotaryInserter.Drive.PLS.Pos2.HighLimit := 0.0;
   RotaryInserter.Drive.PLS.Pos2.Ok := FALSE;
   RotaryInserter.Drive.PLS.Pos3.LowLimit := 0.0;
   RotaryInserter.Drive.PLS.Pos3.HighLimit := 0.0;
   RotaryInserter.Drive.PLS.Pos3.Ok := FALSE;
   RotaryInserter.Drive.PLS.Pos4.LowLimit := 0.0;
   RotaryInserter.Drive.PLS.Pos4.HighLimit := 0.0;
   RotaryInserter.Drive.PLS.Pos4.Ok := FALSE;
   RotaryInserter.Drive.PLS.Pos5.LowLimit := 0.0;
   RotaryInserter.Drive.PLS.Pos5.HighLimit := 0.0;
   RotaryInserter.Drive.PLS.Pos5.Ok := FALSE;
   RotaryInserter.Drive.TON_EnableDrive.PT := T#500MS;
   RotaryInserter.Drive.TON_EnableDrive.IN := FALSE;
   RotaryInserter.Drive.TON_HwOvertravel_Dis.PT := T#0MS;
   RotaryInserter.Drive.TON_HwOvertravel_Dis.IN := FALSE;
   RotaryInserter.Drive.TON_HwOvertravel_En.PT := T#0MS;
   RotaryInserter.Drive.TON_HwOvertravel_En.IN := FALSE;
   RotaryInserter.Drive.TON_TimeoutMovement.PT := T#8S;
   RotaryInserter.Drive.TON_TimeoutMovement.IN := FALSE;
   RotaryInserter.TON_ResetMinLevel.PT := T#2S;
   RotaryInserter.TON_ResetMinLevel.ET := T#2S;
   RotaryInserter.TON_ResetMinLevel.IN := TRUE;
   RotaryInserter.TON_ResetMinLevel.Q := TRUE;
   RotaryInserter.RTO_Work.PT := T#1M;
   RotaryInserter.RTO_Work.IN := FALSE;
   RotaryInserter.TON_ScOK.PT := T#20S;
   RotaryInserter.TON_ScOK.IN := FALSE;
   RotaryInserter.TON_Sign_MinLevel.PT := T#1S;
   RotaryInserter.TON_Sign_MinLevel.IN := FALSE;
   RotaryInserter.TON_TimeoutWork.PT := T#20S;
   RotaryInserter.TON_TimeoutWork.IN := FALSE;
   RotaryInserter.TON_MouldAbsence.PT := T#200MS;
   RotaryInserter.TON_MouldAbsence.IN := FALSE;
   OrientationDetector.AlmOk := FALSE;
   OrientationDetector.CheckMouldHeight := FALSE;
   OrientationDetector.LowMouldHeight := FALSE;
   OrientationDetector.StrobeHeightOk := FALSE;
   OrientationDetector.MouldHeight := 30.0;
   OrientationDetector.Input.MouHeiPrb.EngValue := 0.0;
   OrientationDetector.Input.MouHeiPrb.ScaledValue := 0.0;
   OrientationDetector.Man.Ons_SingleCycle := FALSE;
   OrientationDetector.Man.CmdSingleCycle := FALSE;
   OrientationDetector.Man.EnaPbt := FALSE;
   OrientationDetector.Man.RstCmd := FALSE;
   OrientationDetector.Man.ScreenNumber := 302_100_301;
   OrientationDetector.Man.WithinScreenRange := 0;
   OrientationDetector.TON_CheckMouldHeight.PT := T#500MS;
   OrientationDetector.TON_CheckMouldHeight.IN := FALSE;
END_DATA_BLOCK
